// TIA Portal V20 export
// export: Created 2026-04-10T22:01:57.8344067Z, ExportSetting WithDefaults, DisplayName Totally Integrated Automation Portal, DisplayVersion V20, DisplayName TIA Portal Openness, DisplayVersion V20, DisplayName TIA Portal Version Control Interface, DisplayVersion V20, DisplayName STEP 7 Professional, DisplayVersion V20, DisplayName STEP 7 Safety, DisplayVersion V20, DisplayName WinCC Basic/Comfort/Advanced, DisplayVersion V20
VAR_GLOBAL   // PLC tag table "ELE_"
END_VAR
VAR_GLOBAL CONSTANT   // user constants
   ELE_DRIVE_1 : Int := 1;   // Kommentar ELE_DRIVE_1
   ELE_DRIVE_2 : Int := 2;   // Kommentar ELE_DRIVE_2
   ELE_GENERAL : Int := 3;   // Kommentar ELE_GENERAL
END_VAR
